// TIA Portal V19 export
TYPE "lexchangetray_typeUnEmn_toConstraintWorkstationRecieve"
// Type: lexchangetray_typeconstraintWorkstationEm_toConstraintRollerReq
// Type: lexchangetray_typeconstraintWorkstationEm_toConstraintRollerFeedback
// stored: Access Published
   STRUCT
      feedback : "lexchangetray_typeconstraintWorkstationEm_toConstraintRollerFeedback";
      req : "lexchangetray_typeconstraintWorkstationEm_toConstraintRollerReq";
   END_STRUCT;
END_TYPE
